Staubli VAL3: libDialogs.pjx

--- libDialogs.pjx ---
Parameters version=s7.9.2 stackSize=5000 millimeterUnit=true
Program file=bDialogYesNo.pgx
Program file=clrscr.pgx
Program file=DialogOKandBI.pgx
Program file=DialogOnlyBI.pgx
Program file=DialogOnlyOK.pgx
Program file=nDialogChoices.pgx
Program file=nDialogInsNum.pgx
Program file=sCenterRow.pgx
Program file=sCenterString.pgx
Program file=sCenterTitle.pgx
Program file=teachPoint.pgx
Program file=trsfDialogIns.pgx
Data file=libDialogs.dtx
Library alias=uPage path=./userPage/userPage.pjx

--- libDialogs.dtx ---
string VERSION = "0.3.1"

--- bDialogYesNo.pgx ---
public program bDialogYesNo(string x_sTitle, string x_sQuestion_r1, string x_sQuestion_r2, string x_sQuestion_r3, bool& x_bResp)
  local bool l_bLoop
  local num l_nNum
begin

  //return by using the bResp parameter true if the choose was "yes", false if the choose was "no"
  //notes: screen size is 13rowsX40columns
  //usage: call bDialogYesNo(bRes, "RETURN IN HOME", "ATTENTION:", "Robot will return in home position", "continue?")

  wait(getKey()==-1)

  userPage()
  call clrscr()

  call sCenterTitle(x_sTitle)

  title(x_sTitle)

  gotoxy(0,4)
  call sCenterRow(x_sQuestion_r1)
  putln(x_sQuestion_r1)

  gotoxy(0,5)
  call sCenterRow(x_sQuestion_r2)
  putln(x_sQuestion_r2)

  gotoxy(0,6)
  call sCenterRow(x_sQuestion_r3)
  putln(x_sQuestion_r3)

  gotoxy(0,13)
  put("F1=No")
  gotoxy(34,13)
  put("F8=Yes")

  do
    l_nNum=get()
    if l_nNum==271
      x_bResp=false
    elseIf l_nNum==278
      x_bResp=true
    endIf
  until l_nNum==271 or l_nNum==278

  call clrscr()

  wait(getKey()==-1)

end

--- clrscr.pgx ---
public program clrscr()
begin
  cls()
  title("")
end

--- DialogOKandBI.pgx ---
public program dialogOKandBI(dio x_diBreakInput, string x_sTitle, string x_sText_r1, string x_sText_r2, string x_sText_r3, string x_sText_r4)
  local num l_nNum
begin

  //notes: screen size is 13rowsX40columns
 //usage: call DialogOnlyBI(diStartButton, "START PROGRAM", "Press Start Button or F1", "to start the program", "", "", sUserScreen)

  wait(getKey()==-1)
  userPage()
  call clrscr()

  call sCenterTitle(x_sTitle)

  title(x_sTitle)

  gotoxy(0,4)
  call sCenterRow(x_sText_r1)
  putln(x_sText_r1)

  gotoxy(0,5)
  call sCenterRow(x_sText_r2)
  putln(x_sText_r2)

  gotoxy(0,6)
  call sCenterRow(x_sText_r3)
  putln(x_sText_r3)

  gotoxy(0,7)
  call sCenterRow(x_sText_r4)
  putln(x_sText_r4)

  gotoxy(0,13)
  put("F1=Ok")

  getKey()
  do
    l_nNum=getKey()
    delay(0)
  until l_nNum==271 or x_diBreakInput==true

  call clrscr()
  wait(getKey()==-1)

end

--- DialogOnlyBI.pgx ---
public program dialogOnlyBI(dio x_diBreakInput, string x_sTitle, string x_sText_r1, string x_sText_r2, string x_sText_r3, string x_sText_r4)
  local num l_nNum
begin

  //notes: screen size is 13rowsX40columns
  //usage: call DialogOnlyBI(diStartButton, "START PROGRAM", "Press Start Button", "to start the program", "", "", sUserScreen)

  wait(getKey()==-1)
  userPage()
  call clrscr()

  call sCenterTitle(x_sTitle)

  title(x_sTitle)

  gotoxy(0,4)
  call sCenterRow(x_sText_r1)
  putln(x_sText_r1)

  gotoxy(0,5)
  call sCenterRow(x_sText_r2)
  putln(x_sText_r2)

  gotoxy(0,6)
  call sCenterRow(x_sText_r3)
  putln(x_sText_r3)

  gotoxy(0,7)
  call sCenterRow(x_sText_r4)
  putln(x_sText_r4)

  wait(x_diBreakInput==true)
  call clrscr()
  wait(getKey()==-1)

end

--- DialogOnlyOK.pgx ---
public program dialogOnlyOK(string x_sTitle, string x_sText_r1, string x_sText_r2, string x_sText_r3, string x_sText_r4)
  local num l_nNum
begin

  //notes: screen size is 13rowsX40columns
  //usage: call DialogOnlyOK("RETURN IN HOME", "ATTENTION:", "Robot will return in home position", "be careful!", "", sUserScreen)

  wait(getKey()==-1)
  userPage()
  call clrscr()

  call sCenterTitle(x_sTitle)

  title(x_sTitle)

  gotoxy(0,4)
  call sCenterRow(x_sText_r1)
  putln(x_sText_r1)

  gotoxy(0,5)
  call sCenterRow(x_sText_r2)
  putln(x_sText_r2)

  gotoxy(0,6)
  call sCenterRow(x_sText_r3)
  putln(x_sText_r3)

  gotoxy(0,7)
  call sCenterRow(x_sText_r4)
  putln(x_sText_r4)

  gotoxy(0,13)
  put("F1=Ok")

  do
    l_nNum=get()
  until l_nNum==271

//  getKey()
//  while (getKey()!=271)
//    delay(0)
//  endWhile

  call clrscr()
  wait(getKey()==-1)

end

--- nDialogChoices.pgx ---
public program nDialogChoices(string x_sTitle, string x_sOpt_r1, string x_sOpt_r2, string x_sOpt_r3, string x_sOpt_r4, string x_sOpt_r5, string x_sOpt_r6, num& x_nResp)
  local num l_nNum
  local bool l_bLoop
begin

  //return by using the nResp parameter the index of the option choosed
  //notes: screen size is 13rowsX40columns
  //usage: ...set as "" every option you don't need to use example:
  //call nDialogChoices("MULTIPLE OPTIONS", "option1", "option2", "", "option4", "option5", "option6", nResp)

  wait(getKey()==-1)
  userPage()
  call clrscr()

  call sCenterTitle(x_sTitle)

  title(x_sTitle)

  if x_sOpt_r1!=""
    gotoxy(0,2)
    //call sCenterRow(x_sOpt_r1)
    put("F1-->")
    putln(x_sOpt_r1)
  endIf

  if x_sOpt_r2!=""
    gotoxy(0,3)
    //call sCenterRow(x_sOpt_r2)
    put("F2-->")
    putln(x_sOpt_r2)
  endIf

  if x_sOpt_r3!=""
    gotoxy(0,4)
    //call sCenterRow(x_sOpt_r3)
    put("F3-->")
    putln(x_sOpt_r3)
  endIf

  if x_sOpt_r4!=""
    gotoxy(0,5)
    //call sCenterRow(x_sOpt_r4)
    put("F4-->")
    putln(x_sOpt_r4)
  endIf

  if x_sOpt_r5!=""
    gotoxy(0,6)
    //call sCenterRow(x_sOpt_r5)
    put("F5-->")
    putln(x_sOpt_r5)
  endIf

  if x_sOpt_r6!=""
    gotoxy(0,7)
    //call sCenterRow(x_sOpt_r5)
    put("F6-->")
    putln(x_sOpt_r6)
  endIf


  getKey()
  l_bLoop=true

  while l_bLoop
    l_nNum=get()
    if l_nNum==271 and x_sOpt_r1!=""
      x_nResp=0
      l_bLoop=false
    elseIf l_nNum==272 and x_sOpt_r2!=""
      x_nResp=1
      l_bLoop=false
    elseIf l_nNum==273 and x_sOpt_r3!=""
      x_nResp=2
      l_bLoop=false
    elseIf l_nNum==274 and x_sOpt_r4!=""
      x_nResp=3
      l_bLoop=false
    elseIf l_nNum==275 and x_sOpt_r5!=""
      x_nResp=4
      l_bLoop=false
    elseIf l_nNum==276 and x_sOpt_r6!=""
      x_nResp=5
      l_bLoop=false
    endIf
  endWhile

  call clrscr()
  wait(getKey()==-1)

end

--- nDialogInsNum.pgx ---
public program nDialogInsNum(string x_sTitle, string x_sText_r1, num& x_nNum)
  local num l_nVal
  local num l_nKey
begin

  //notes: screen size is 13rowsX40columns
  //usage: call DialogInsNums("NUMERIC INS", "Insert a value for foo:", num, screen)

  wait(getKey()==-1)
  userPage()
  call clrscr()
  l_nVal=x_nNum


  call sCenterTitle(x_sTitle)

  title(x_sTitle)

  gotoxy(0,4)
  //call sCenterRow(x_sText_r1)
  put(x_sText_r1)

  gotoxy(34,13)
  put("F8=Ok")

  gotoxy(0,13)
  put("F1=Esc")

  gotoxy(len(x_sText_r1)+1,4)
  gotoxy(len(x_sText_r1)+1, 4)


  do
    l_nKey=get(l_nVal)
    if l_nKey==278
      x_nNum=l_nVal
    endIf
  until l_nKey==271 or l_nKey==278

  call clrscr()
  wait(getKey()==-1)

end

--- sCenterRow.pgx ---
program sCenterRow(string& x_sRow)
begin

  //max length 40 characters
  call sCenterString(x_sRow,asc(" ",0),40)

end

--- sCenterString.pgx ---
program sCenterString(string& x_sString, num x_nFillerAsc, num x_nMaxLength)
  local num l_nIndex_i
  local string l_sLeadingSpa
  local string l_sTrailingSpa
begin

  x_sString=left(x_sString,x_nMaxLength)

  //adding spaces to centre the string
  for l_nIndex_i=0 to roundDown((x_nMaxLength-len(x_sString)-1)/2)
    l_sLeadingSpa=l_sLeadingSpa+chr(x_nFillerAsc)
    l_sTrailingSpa=l_sTrailingSpa+chr(x_nFillerAsc)
  endFor

  x_sString=l_sLeadingSpa+x_sString+l_sTrailingSpa

  x_sString=left(x_sString,x_nMaxLength)

end

--- sCenterTitle.pgx ---
public program sCenterTitle(string& x_sTitle)
  local num l_nIndex_i
  local string l_sLeadingSpa
  local string l_sTrailingSpa
begin


  //max length 36 characters
  call sCenterString(x_sTitle,asc("=",0),36)


end

--- teachPoint.pgx ---
public program teachPoint(string x_sPointName, tool x_tTool, frame x_fFrame, point& x_pPoint)
  local string l_sTemp
  local num l_nNum
  local point l_pPoint
begin

  wait(getKey()==-1)

  userPage()
  call clrscr()

  l_sTemp = "teaching "+x_sPointName
  call sCenterTitle(l_sTemp)

  title(l_sTemp)

  gotoxy(0,4)
  l_sTemp = "premi F8 per acquisire "+x_sPointName
  call sCenterRow(l_sTemp)
  putln(l_sTemp)

  gotoxy(0,5)
  l_sTemp = "premi F1 per uscire"
  call sCenterRow(l_sTemp)
  putln(l_sTemp)

  gotoxy(0,13)
  put("F1=Esc")
  gotoxy(34,13)
  put("F8=Qui")

  do
    l_nNum=get()
    if l_nNum==271
      call dialogOnlyOK("teaching "+x_sPointName,"acquisizione punto annullata",x_sPointName+" non è stato modificato","premi F1 per continuare","")
    elseIf l_nNum==278
      l_pPoint = here(x_tTool, x_fFrame)
      x_pPoint.trsf = position(l_pPoint, x_fFrame)
      call trsfDialogIns("teaching "+x_sPointName, "", x_pPoint.trsf)
    endIf
  until l_nNum==271 or l_nNum==278

  call clrscr()

  wait(getKey()==-1)

end

--- trsfDialogIns.pgx ---
public program trsfDialogIns(string x_sTitle, string x_sComment, trsf& x_tTrsf)
begin

  call uPage:changeTrsf(x_tTrsf, x_sTitle, x_sComment)
  call clrscr()

end
